SYSTEM Test System
  (* Version 1.0, 2005-06-15, Goran Cengic, Chalmers *)
  DEVICE Test Device : DeviceType_not_used
    RESOURCE TestResource : ResourceType_not_used
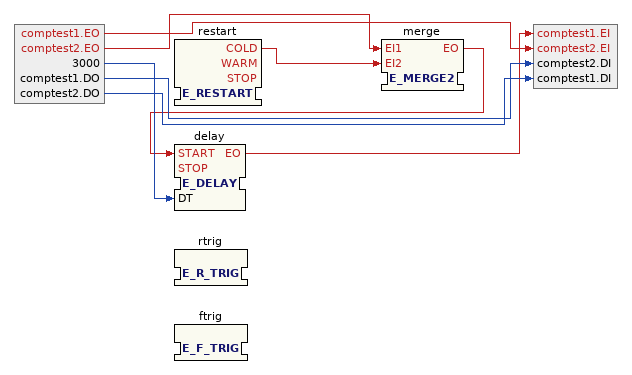
      FBS
        restart : E_RESTART;
        delay : E_DELAY;
        merge : E_MERGE2;
        rtrig : E_R_TRIG;
        ftrig : E_F_TRIG;
      END_FBS
      EVENT_CONNECTIONS
        restart.COLD TO merge.EI2;
        merge.EO TO delay.START;
        delay.EO TO comptest1.EI;
        comptest1.EO TO comptest2.EI;
        comptest2.EO TO merge.EI1;
      END_CONNECTIONS
      DATA_CONNECTIONS
        3000 TO delay.DT;
        comptest1.DO TO comptest2.DI;
        comptest2.DO TO comptest1.DI;
      END_CONNECTIONS
    END_RESOURCE
  END_DEVICE
END_SYSTEM
